TYPE ST_TcpVisionOutCmd :
STRUCT
    JudgeOk   : BOOL;
    ResultData: STRING(255);
END_STRUCT
END_TYPE

(* stored: Version 1.1.0.1, ProductVersion 3.1.4024.12
   DUT ST_TcpVisionOutCmd: Id {513dd763-eafc-4894-b237-f08ee6334853} *)
